{region '#Template'}
	{attribute 'Version' := '1.2.0.0'}
	{attribute 'Tags' := '"LCID": "1031", "Text": "DUT, Building, RA, OpMod, Mode"'}
	{attribute 'Tags' := '"LCID": "1033", "Text": "DUT, Building, RA, OpMod, Mode"'}
	{attribute 'Description' := '"LCID": "1031", "Text": "Gebäude-Betriebsart"'}
	{attribute 'Description' := '"LCID": "1033", "Text": "Building-operation-mode"'}
{endregion}

{attribute qualified_only}
TYPE E_BA_BuildingMode :
(
	eDefault		:= 1,
	eNightWatch		:= 2,
	eCleaning		:= 3
	
) UDINT;
END_TYPE

(* stored: Version 1.1.0.1, ProductVersion 3.1.4024.9
   DUT E_BA_BuildingMode: Id {dfdb4296-b0b9-4d72-9317-b405c599d365} *)
